PROGRAM PendantControl
VAR
	Selection: UINT;
	Cover3_state: RS;
	Cover3_axis: 		MDP5001_511_733_5131DD77;
	Cover3_control:		FB_DCAxis;
	Cover2_axis: 		MDP5001_511_733_5131DD77;
	Cover2_control:		FB_DCAxis;
	Nasmyth_axis:		MDP5001_511_733_5131DD77;
	Nasmyth_control:	FB_DCAxis;
	error:				BOOL;
	Nasmyth_delay:		TON;
	Nasmyth_unlock,
	Nasmyth_unlocked:	BOOL;
	DerotatorAxisJog:	FB_AxisJog;
	//AzimuthAxisJog:		FB_AxisJog;
	Focus_enable,
	Elevation_enable,
	Azimuth_enable,
	Dome_enable,
	FilterWheel_enable : BOOL := FALSE;
	manual,
	enable,
	reset,
	up,
	down,
	left,
	right,
	manual_hydraulics_start,
	manual_hydraulics_stop:		BOOL;
	
	brake_state:	RS;
	brake_open : BOOL;
END_VAR

Selection := 1*BOOL_TO_UINT(GVL_pendant_control.BCD1) + 
			 2*BOOL_TO_UINT(GVL_pendant_control.BCD2) + 
			 4*BOOL_TO_UINT(GVL_pendant_control.BCD4) +
			 8*BOOL_TO_UINT(GVL_pendant_control.BCD8);

GVL_pendant_control.lamp_left := FALSE;
GVL_pendant_control.lamp_right := FALSE;
GVL_pendant_control.lamp_up := FALSE;
GVL_pendant_control.lamp_down := FALSE;
manual := GVL_pendant_control.key_switch;
enable := GVL_pendant_control.start_switch;
reset := GVL_pendant_control.reset_switch;
up := GVL_pendant_control.direction_up;
down := GVL_pendant_control.direction_down;
left := GVL_pendant_control.direction_left;
right := GVL_pendant_control.direction_right;

GVL_pendant_control.lamp_error := GVL_Main.lamp_error;

IF NOT manual THEN 
	// we have nothing to do further
	RETURN;
END_IF;

Nasmyth_delay(IN := GVL_Telescope.nasmyth_lock,
				PT := T#500MS,
				Q => Nasmyth_unlocked);

Focus_enable := FALSE;
Elevation_enable := FALSE;
Azimuth_enable := FALSE;
Dome_enable := FALSE;
FilterWheel_enable := FALSE;

CASE Selection OF
	1:	GVL_pendant_control.lamp_left := TRUE;
		GVL_pendant_control.lamp_right := TRUE;
	2: Cover2_control(open := up,
						close := down,
						enable := manual AND GVL_Telescope.cover3_closed,
						reset := MAIN.reset,
						limit_open := GVL_Telescope.cover2_open,
						limit_close := GVL_Telescope.cover2_closed,
						error => error,
						axis_ref := Cover2_axis);
		GVL_pendant_control.lamp_up := GVL_Telescope.cover2_open;
		GVL_pendant_control.lamp_down := GVL_Telescope.cover2_closed;
 
	
	3:  
		 Cover3_control(open := up,
						close := down,
						enable := manual,
						reset := MAIN.reset,
						limit_open := GVL_Telescope.cover3_open,
						limit_close := GVL_Telescope.cover3_closed,
						error => error,
						axis_ref := Cover3_axis);
		GVL_pendant_control.lamp_up := GVL_Telescope.cover3_open;
		GVL_pendant_control.lamp_down := GVL_Telescope.cover3_closed;
	4:
		GVL_Telescope.nasmyth_lock :=  manual AND 
										( left OR 
 										right OR
										enable);
										
		 Nasmyth_control(open := left AND Nasmyth_unlocked,
						close := right AND Nasmyth_unlocked,
						enable := GVL_pendant_control.key_switch,
						reset := MAIN.reset,
						limit_open := NOT GVL_Telescope.nasmyth_limit_right,
						limit_close := NOT GVL_Telescope.nasmyth_limit_left,
						error => error,
						velocity := 18000,
						axis_ref := Nasmyth_axis);
		GVL_pendant_control.lamp_left := GVL_Telescope.nasmyth_limit_left;
		GVL_pendant_control.lamp_right := GVL_Telescope.nasmyth_limit_right;
		
	5:	GVL_pendant_control.lamp_up := NOT GVL_Telescope.focus_limit_far;
		GVL_pendant_control.lamp_down := NOT GVL_Telescope.focus_limit_near;
		Focus_enable := manual;
		FocusControl.outward := up;
		FocusControl.inward := down;
		Focuscontrol.reset := reset;
						
	6:	GVL_pendant_control.lamp_left := TRUE;
		GVL_pendant_control.lamp_right := TRUE;
		DeRotatorAxisJog(bPowerEnable := manual AND Main.power_OK,
						bEnable_Positive := TRUE,
						bEnable_Negative := TRUE,
						bForward := right,
						bBackward := left,
						bReset := manual AND reset,
						bStop := manual AND enable,
						bErr => error,
						stAxis :=	GVL_Telescope.DerotatorAxisRef);
						
	7:	Elevation_enable := manual;
		GVL_pendant_control.lamp_up := Elevation_enable;
		GVL_pendant_control.lamp_down := Elevation_enable;
		ElevationControl.up := up;
		ElevationControl.down := down;
		ElevationControl.reset := reset;
		
	8:	// This selection will become RA/Dec Mode with tracking enabled!
		Azimuth_enable := manual;
		GVL_pendant_control.lamp_left := Azimuth_enable;
		GVL_pendant_control.lamp_right := Azimuth_enable;
		AzimuthControl.left := left;
		AzimuthControl.right := right;
		AzimuthControl.reset := reset;
		
	9: 	Dome_enable := manual;
		GVL_pendant_control.lamp_left := Dome_enable;
		GVL_pendant_control.lamp_right := Dome_enable;
		DomeControl.left := left;
		DomeControl.right := right;
		DomeControl.reset := reset;
		
	10:	FilterWheel_enable := manual;
		GVL_pendant_control.lamp_left := FilterWheel_enable;
		GVL_pendant_control.lamp_right := FilterWheel_enable;
		FilterWheelControl.left := left;
		FilterWheelControl.right := right;
		FilterWheelControl.reset := reset;
	
	15:	GVL_pendant_control.lamp_up := HydraulicsControl.oil_pressure_OK AND NOT brake_open;
		GVL_pendant_control.lamp_down := HydraulicsControl.oil_pressure_OK AND brake_open;
		GVL_pendant_control.lamp_left := HydraulicsControl.pump_running;
		GVL_pendant_control.lamp_right := HydraulicsControl.suction_running;
		manual_hydraulics_start := manual AND enable;
		manual_hydraulics_stop := manual AND reset;
		brake_state(SET := up,
					Reset1 := down,
					Q1 => brake_open);
		
END_CASE

FocusControl.enable := Focus_enable;
ElevationControl.enable := Elevation_enable;
AzimuthControl.enable := Azimuth_enable;
DomeControl.enable := Dome_enable;
FilterWheelControl.enable := FilterWheel_enable;
GVL_pendant_control.lamp_error := Main.error;

END_PROGRAM

(* stored: Version 1.1.0.1, ProductVersion 3.1.4024.4
   POU PendantControl: Id {4c9494b1-b987-44f6-88ae-faae341979f2}, SpecialFunc None *)
